// Mitsubishi GX Works2 project: ladder_dac   PLC: Q02U

PROGRAM MAIN
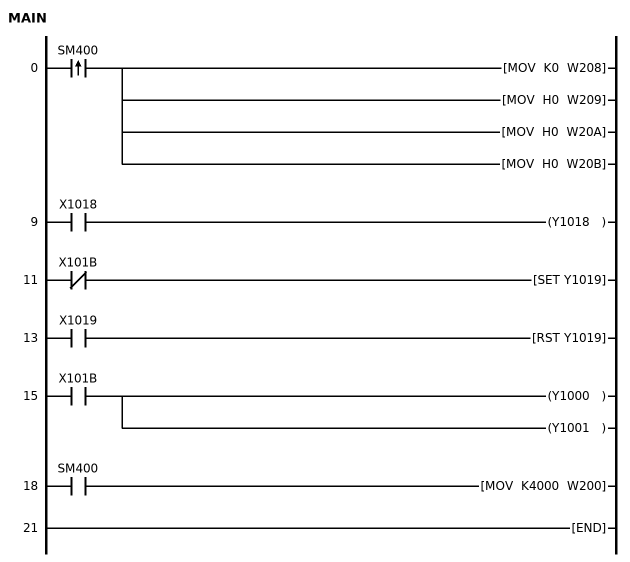
0     LDP     SM400
      MOV     K0 W208
      MOV     H0 W209
      MOV     H0 W20A
      MOV     H0 W20B
9     LD      X1018
      OUT     Y1018
11    LDI     X101B
      SET     Y1019
13    LD      X1019
      RST     Y1019
15    LD      X101B
      OUT     Y1000
      OUT     Y1001
18    LD      SM400
      MOV     K4000 W200
21    END
END_PROGRAM
